// TIA Portal V20 export
DATA_BLOCK "SP502"   // DB340
// stored: MemoryReserve 100
   VAR
      "CLASS2 SMPS ALARM RESET" : Bool := FALSE;
      SPARE_4 : Bool := FALSE;
      SPARE_5 : Bool := FALSE;
      SPARE_6 : Bool := FALSE;
      SPARE_7 : Bool := FALSE;
      SPARE_8 : Bool := FALSE;
      SPARE_9 : Bool := FALSE;
      SPARE_10 : Bool := FALSE;
      "SEPA UW IONIZER TOP MAINTERNANCE DETECTION" : Bool := FALSE;
      "SEPA UW IONIZER TOP DISCHARGE STOP" : Bool := FALSE;
      SPARE : Bool := FALSE;
      SPARE_1 : Bool := FALSE;
      "SEPA UW IONIZER BOTTOM MAINTERNANCE DETECTION" : Bool := FALSE;
      "SEPA UW IONIZER BOTTOM DISCHARGE STOP" : Bool := FALSE;
   END_VAR
BEGIN
END_DATA_BLOCK
